(********************* G.D S.p.A. - Technical Department ***********************************
This program has been generated automatically from Application Designer DE&F
********************************************************************************************)
PROGRAM dbg_csp_transfer_main_safety_guards
VAR
  delayed_sis_shd : safety_integrated_series_shadow;
  sio_door_3_shd : safety_integrated_object_shadow;
  sio_door_4_shd : safety_integrated_object_shadow;
  sio_door_5_shd : safety_integrated_object_shadow;
  sio_door_6_shd : safety_integrated_object_shadow;
  sio_door_7_shd : safety_integrated_object_shadow;
  sio_door_8_shd : safety_integrated_object_shadow;
  sis_shd : safety_integrated_series_shadow;
END_VAR

_objects_manager();

IF	g_application_status <> APPLICATION_STATUS_RUNNING
THEN
	RETURN;
END_IF

CASE process_get_mode(CONVERSION_this := dbg_root.prc) OF
	MODE_ABSENT,
	MODE_INACTIVE:
		RETURN;
	MODE_TEST:
		RETURN;
END_CASE

ACTION _objects_manager:
IF	objects_initialization()
THEN
	safety_integrated_series_shadow_init(
		sim_mode:= SHADOW_SIMULATION_MODE_AUTOMATIC, 
		father:= csp_transfer_main_safety_guards.delayed_sis, 
		process:= dbg_root.prc, 
		CONVERSION_this:= delayed_sis_shd);

	safety_integrated_object_shadow_init(
		sim_mode:= SHADOW_SIMULATION_MODE_AUTOMATIC, 
		father:= csp_transfer_main_safety_guards.sio_door_3, 
		process:= dbg_root.prc, 
		CONVERSION_this:= sio_door_3_shd);

	safety_integrated_object_shadow_init(
		sim_mode:= SHADOW_SIMULATION_MODE_AUTOMATIC, 
		father:= csp_transfer_main_safety_guards.sio_door_4, 
		process:= dbg_root.prc, 
		CONVERSION_this:= sio_door_4_shd);

	safety_integrated_object_shadow_init(
		sim_mode:= SHADOW_SIMULATION_MODE_AUTOMATIC, 
		father:= csp_transfer_main_safety_guards.sio_door_5, 
		process:= dbg_root.prc, 
		CONVERSION_this:= sio_door_5_shd);

	safety_integrated_object_shadow_init(
		sim_mode:= SHADOW_SIMULATION_MODE_AUTOMATIC, 
		father:= csp_transfer_main_safety_guards.sio_door_6, 
		process:= dbg_root.prc, 
		CONVERSION_this:= sio_door_6_shd);

	safety_integrated_object_shadow_init(
		sim_mode:= SHADOW_SIMULATION_MODE_AUTOMATIC, 
		father:= csp_transfer_main_safety_guards.sio_door_7, 
		process:= dbg_root.prc, 
		CONVERSION_this:= sio_door_7_shd);

	safety_integrated_object_shadow_init(
		sim_mode:= SHADOW_SIMULATION_MODE_AUTOMATIC, 
		father:= csp_transfer_main_safety_guards.sio_door_8, 
		process:= dbg_root.prc, 
		CONVERSION_this:= sio_door_8_shd);

	safety_integrated_series_shadow_init(
		sim_mode:= SHADOW_SIMULATION_MODE_AUTOMATIC, 
		father:= csp_transfer_main_safety_guards.sis, 
		process:= dbg_root.prc, 
		CONVERSION_this:= sis_shd);

	RETURN;
END_IF

IF	objects_running()
THEN
	safety_integrated_series_shadow_cycle(delayed_sis_shd);
	safety_integrated_object_shadow_cycle(sio_door_3_shd);
	safety_integrated_object_shadow_cycle(sio_door_4_shd);
	safety_integrated_object_shadow_cycle(sio_door_5_shd);
	safety_integrated_object_shadow_cycle(sio_door_6_shd);
	safety_integrated_object_shadow_cycle(sio_door_7_shd);
	safety_integrated_object_shadow_cycle(sio_door_8_shd);
	safety_integrated_series_shadow_cycle(sis_shd);
END_IF
END_ACTION

END_PROGRAM

(* stored: Version 1.1.0.1, ProductVersion 3.1.4022.12
   POU dbg_csp_transfer_main_safety_guards: Id {4ff63161-0171-49e0-8cd0-f312c75dbd1e}, SpecialFunc None
   Action _objects_manager: Id {00c9d6bf-3bd1-4dcb-9055-45af6dff2a92} *)
